// Mitsubishi GX Works2 project: indexing   PLC: Q02/Q02H

PROGRAM MAIN
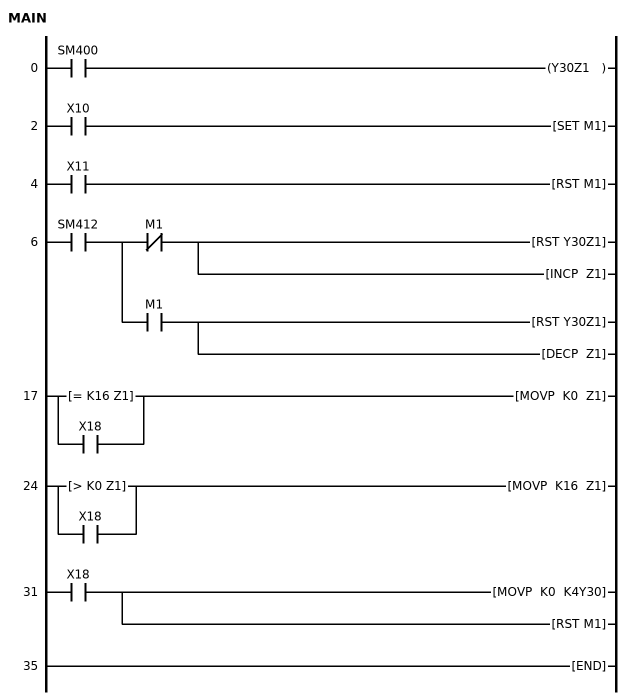
0     LD      SM400
      OUT     Y30Z1
2     LD      X10
      SET     M1
4     LD      X11
      RST     M1
6     LD      SM412
      MPS
      ANI     M1
      RST     Y30Z1
      INCP    Z1
      MPP
      AND     M1
      RST     Y30Z1
      DECP    Z1
17    LD=     K16 Z1
      OR      X18
      MOVP    K0 Z1
24    LD>     K0 Z1
      OR      X18
      MOVP    K16 Z1
31    LD      X18
      MOVP    K0 K4Y30
      RST     M1
35    END
END_PROGRAM

PROGRAM MAIN2
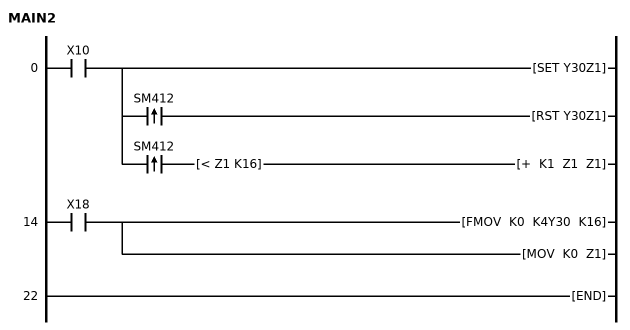
0     LD      X10
      SET     Y30Z1
      MPS
      ANDP    SM412
      RST     Y30Z1
      MPP
      ANDP    SM412
      AND<    Z1 K16
      +       K1 Z1 Z1
14    LD      X18
      FMOV    K0 K4Y30 K16
      MOV     K0 Z1
22    END
END_PROGRAM

PROGRAM MAIN1
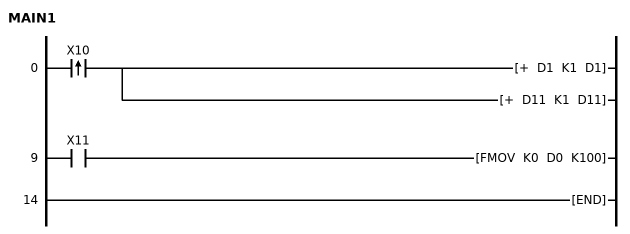
0     LDP     X10
      +       D1 K1 D1
      +       D11 K1 D11
9     LD      X11
      FMOV    K0 D0 K100
14    END
END_PROGRAM
